{attribute 'pack_mode' := '2'}
TYPE ST_DATA_STATE :
STRUCT
  State       : E_DATA_STATE;
  Init        : E_PROGRESS;
END_STRUCT
END_TYPE

(* stored: Version 1.1.0.1, ProductVersion 3.1.4026.18
   DUT ST_DATA_STATE: Id {7681e77f-cdf7-4acf-a944-d1bee289acea} *)
